// TIA Portal V20 export
TYPE "LBP_typeNCVariableTokenUInt"
TITLE = LBP_ReadVar and LBP_WriteVar Interface / Interface LBP_ReadVar et LBP_WriteVar
// User Data Type for LBP_ReadVar[FB2] and LBP_WriteVar[FB3] Parameters / Type de données utilisateur pour les paramètres LBP_ReadVar[FB2] et LBP_WriteVar[FB3]
   STRUCT
      token : "LBP_typeNCVariableToken";   // User Data Type for LBP_ReadVar[FB2] and LBP_WriteVar[FB3] Input Parameter Addrx / Type de données utilisateur pour les paramètres d'entrée Addrx LBP_ReadVar[FB2] et LBP_WriteVar[FB3]
      value : UInt;   // Data Type for LBP_ReadVar[FB2] and LBP_WriteVar[FB3] InOut Parameter SDx / Type de données pour les paramètres E/S SDx LBP_ReadVar[FB2] et LBP_WriteVar[FB3]
   END_STRUCT;
END_TYPE
